// TIA Portal V21 export
FUNCTION_BLOCK "Inputs_FB"   // FB100, LAD
{ S7_Optimized_Access := 'TRUE' }
// stored: AutoNumber false, MemoryReserve 100, SetENOAutomatically false
   VAR
      ResetEdge { ExternalAccessible := 'False'; ExternalVisible := 'False'; ExternalWritable := 'False'} : Bool;
      TankLevel { ExternalAccessible := 'False'; ExternalVisible := 'False'; ExternalWritable := 'False'} : Array[1..2] of "AnalogInput";
   END_VAR
   VAR_TEMP   // added for the SCL form of the ladder/FBD networks
      _w1 : Bool;
      _w2 : Bool;
   END_VAR
BEGIN

REGION Network 1: === General
END_REGION

REGION Network 2: Emergency stop
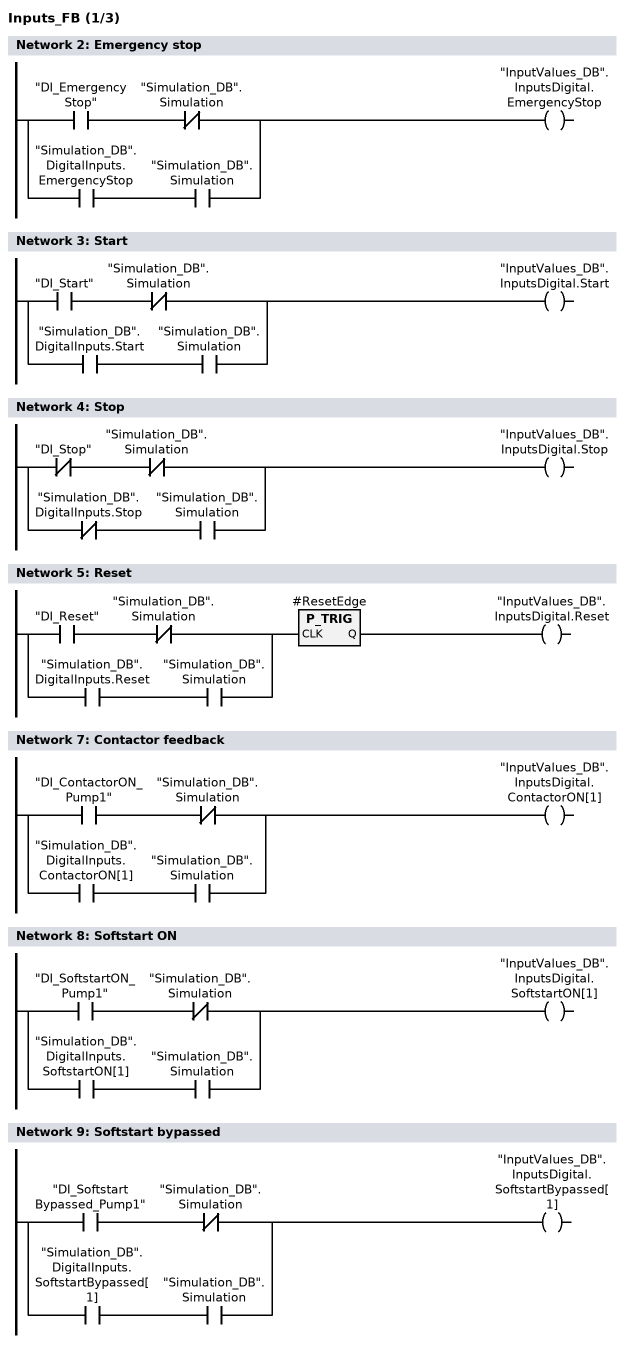
   RUNG wire#powerrail
      Contact( "DI_EmergencyStop" )
      I_Contact( "Simulation_DB".Simulation )
      wire#w1
      Coil( "InputValues_DB".InputsDigital.EmergencyStop )
   END_RUNG
   RUNG wire#powerrail
      Contact( "Simulation_DB".DigitalInputs.EmergencyStop )
      Contact( "Simulation_DB".Simulation )
   END_RUNG wire#w1
   // the same network as SCL:
   "InputValues_DB".InputsDigital.EmergencyStop := ("DI_EmergencyStop" AND NOT "Simulation_DB".Simulation) OR ("Simulation_DB".DigitalInputs.EmergencyStop AND "Simulation_DB".Simulation);
END_REGION

REGION Network 3: Start
   RUNG wire#powerrail
      Contact( "DI_Start" )
      I_Contact( "Simulation_DB".Simulation )
      wire#w1
      Coil( "InputValues_DB".InputsDigital.Start )
   END_RUNG
   RUNG wire#powerrail
      Contact( "Simulation_DB".DigitalInputs.Start )
      Contact( "Simulation_DB".Simulation )
   END_RUNG wire#w1
   // the same network as SCL:
   "InputValues_DB".InputsDigital.Start := ("DI_Start" AND NOT "Simulation_DB".Simulation) OR ("Simulation_DB".DigitalInputs.Start AND "Simulation_DB".Simulation);
END_REGION

REGION Network 4: Stop
   RUNG wire#powerrail
      I_Contact( "DI_Stop" )
      I_Contact( "Simulation_DB".Simulation )
      wire#w1
      Coil( "InputValues_DB".InputsDigital.Stop )
   END_RUNG
   RUNG wire#powerrail
      I_Contact( "Simulation_DB".DigitalInputs.Stop )
      Contact( "Simulation_DB".Simulation )
   END_RUNG wire#w1
   // the same network as SCL:
   "InputValues_DB".InputsDigital.Stop := (NOT "DI_Stop" AND NOT "Simulation_DB".Simulation) OR (NOT "Simulation_DB".DigitalInputs.Stop AND "Simulation_DB".Simulation);
END_REGION

REGION Network 5: Reset
   RUNG wire#powerrail
      Contact( "DI_Reset" )
      I_Contact( "Simulation_DB".Simulation )
      wire#w1
      P_Trig( #ResetEdge )
      Coil( "InputValues_DB".InputsDigital.Reset )
   END_RUNG
   RUNG wire#powerrail
      Contact( "Simulation_DB".DigitalInputs.Reset )
      Contact( "Simulation_DB".Simulation )
   END_RUNG wire#w1
   // the same network as SCL:
   #_w1 := ("DI_Reset" AND NOT "Simulation_DB".Simulation) OR ("Simulation_DB".DigitalInputs.Reset AND "Simulation_DB".Simulation);
   #_w2 := #_w1 AND NOT #ResetEdge;   // rising edge
   #ResetEdge := #_w1;
   "InputValues_DB".InputsDigital.Reset := #_w2;
END_REGION

REGION Network 6: === Pump 1
END_REGION

REGION Network 7: Contactor feedback
   RUNG wire#powerrail
      Contact( "DI_ContactorON_Pump1" )
      I_Contact( "Simulation_DB".Simulation )
      wire#w1
      Coil( "InputValues_DB".InputsDigital.ContactorON[1] )
   END_RUNG
   RUNG wire#powerrail
      Contact( "Simulation_DB".DigitalInputs.ContactorON[1] )
      Contact( "Simulation_DB".Simulation )
   END_RUNG wire#w1
   // the same network as SCL:
   "InputValues_DB".InputsDigital.ContactorON[1] := ("DI_ContactorON_Pump1" AND NOT "Simulation_DB".Simulation) OR ("Simulation_DB".DigitalInputs.ContactorON[1] AND "Simulation_DB".Simulation);
END_REGION

REGION Network 8: Softstart ON
   RUNG wire#powerrail
      Contact( "DI_SoftstartON_Pump1" )
      I_Contact( "Simulation_DB".Simulation )
      wire#w1
      Coil( "InputValues_DB".InputsDigital.SoftstartON[1] )
   END_RUNG
   RUNG wire#powerrail
      Contact( "Simulation_DB".DigitalInputs.SoftstartON[1] )
      Contact( "Simulation_DB".Simulation )
   END_RUNG wire#w1
   // the same network as SCL:
   "InputValues_DB".InputsDigital.SoftstartON[1] := ("DI_SoftstartON_Pump1" AND NOT "Simulation_DB".Simulation) OR ("Simulation_DB".DigitalInputs.SoftstartON[1] AND "Simulation_DB".Simulation);
END_REGION

REGION Network 9: Softstart bypassed
   RUNG wire#powerrail
      Contact( "DI_SoftstartBypassed_Pump1" )
      I_Contact( "Simulation_DB".Simulation )
      wire#w1
      Coil( "InputValues_DB".InputsDigital.SoftstartBypassed[1] )
   END_RUNG
   RUNG wire#powerrail
      Contact( "Simulation_DB".DigitalInputs.SoftstartBypassed[1] )
      Contact( "Simulation_DB".Simulation )
   END_RUNG wire#w1
   // the same network as SCL:
   "InputValues_DB".InputsDigital.SoftstartBypassed[1] := ("DI_SoftstartBypassed_Pump1" AND NOT "Simulation_DB".Simulation) OR ("Simulation_DB".DigitalInputs.SoftstartBypassed[1] AND "Simulation_DB".Simulation);
END_REGION

REGION Network 10: Softstart fault
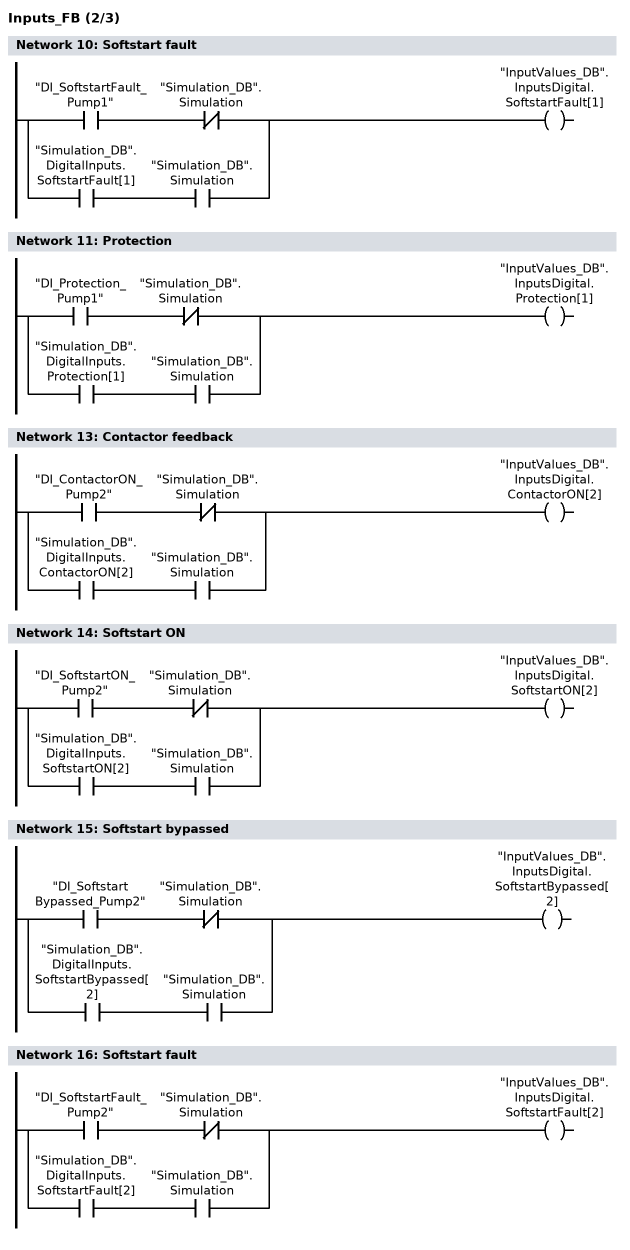
   RUNG wire#powerrail
      Contact( "DI_SoftstartFault_Pump1" )
      I_Contact( "Simulation_DB".Simulation )
      wire#w1
      Coil( "InputValues_DB".InputsDigital.SoftstartFault[1] )
   END_RUNG
   RUNG wire#powerrail
      Contact( "Simulation_DB".DigitalInputs.SoftstartFault[1] )
      Contact( "Simulation_DB".Simulation )
   END_RUNG wire#w1
   // the same network as SCL:
   "InputValues_DB".InputsDigital.SoftstartFault[1] := ("DI_SoftstartFault_Pump1" AND NOT "Simulation_DB".Simulation) OR ("Simulation_DB".DigitalInputs.SoftstartFault[1] AND "Simulation_DB".Simulation);
END_REGION

REGION Network 11: Protection
   RUNG wire#powerrail
      Contact( "DI_Protection_Pump1" )
      I_Contact( "Simulation_DB".Simulation )
      wire#w1
      Coil( "InputValues_DB".InputsDigital.Protection[1] )
   END_RUNG
   RUNG wire#powerrail
      Contact( "Simulation_DB".DigitalInputs.Protection[1] )
      Contact( "Simulation_DB".Simulation )
   END_RUNG wire#w1
   // the same network as SCL:
   "InputValues_DB".InputsDigital.Protection[1] := ("DI_Protection_Pump1" AND NOT "Simulation_DB".Simulation) OR ("Simulation_DB".DigitalInputs.Protection[1] AND "Simulation_DB".Simulation);
END_REGION

REGION Network 12: === Pump 2
END_REGION

REGION Network 13: Contactor feedback
   RUNG wire#powerrail
      Contact( "DI_ContactorON_Pump2" )
      I_Contact( "Simulation_DB".Simulation )
      wire#w1
      Coil( "InputValues_DB".InputsDigital.ContactorON[2] )
   END_RUNG
   RUNG wire#powerrail
      Contact( "Simulation_DB".DigitalInputs.ContactorON[2] )
      Contact( "Simulation_DB".Simulation )
   END_RUNG wire#w1
   // the same network as SCL:
   "InputValues_DB".InputsDigital.ContactorON[2] := ("DI_ContactorON_Pump2" AND NOT "Simulation_DB".Simulation) OR ("Simulation_DB".DigitalInputs.ContactorON[2] AND "Simulation_DB".Simulation);
END_REGION

REGION Network 14: Softstart ON
   RUNG wire#powerrail
      Contact( "DI_SoftstartON_Pump2" )
      I_Contact( "Simulation_DB".Simulation )
      wire#w1
      Coil( "InputValues_DB".InputsDigital.SoftstartON[2] )
   END_RUNG
   RUNG wire#powerrail
      Contact( "Simulation_DB".DigitalInputs.SoftstartON[2] )
      Contact( "Simulation_DB".Simulation )
   END_RUNG wire#w1
   // the same network as SCL:
   "InputValues_DB".InputsDigital.SoftstartON[2] := ("DI_SoftstartON_Pump2" AND NOT "Simulation_DB".Simulation) OR ("Simulation_DB".DigitalInputs.SoftstartON[2] AND "Simulation_DB".Simulation);
END_REGION

REGION Network 15: Softstart bypassed
   RUNG wire#powerrail
      Contact( "DI_SoftstartBypassed_Pump2" )
      I_Contact( "Simulation_DB".Simulation )
      wire#w1
      Coil( "InputValues_DB".InputsDigital.SoftstartBypassed[2] )
   END_RUNG
   RUNG wire#powerrail
      Contact( "Simulation_DB".DigitalInputs.SoftstartBypassed[2] )
      Contact( "Simulation_DB".Simulation )
   END_RUNG wire#w1
   // the same network as SCL:
   "InputValues_DB".InputsDigital.SoftstartBypassed[2] := ("DI_SoftstartBypassed_Pump2" AND NOT "Simulation_DB".Simulation) OR ("Simulation_DB".DigitalInputs.SoftstartBypassed[2] AND "Simulation_DB".Simulation);
END_REGION

REGION Network 16: Softstart fault
   RUNG wire#powerrail
      Contact( "DI_SoftstartFault_Pump2" )
      I_Contact( "Simulation_DB".Simulation )
      wire#w1
      Coil( "InputValues_DB".InputsDigital.SoftstartFault[2] )
   END_RUNG
   RUNG wire#powerrail
      Contact( "Simulation_DB".DigitalInputs.SoftstartFault[2] )
      Contact( "Simulation_DB".Simulation )
   END_RUNG wire#w1
   // the same network as SCL:
   "InputValues_DB".InputsDigital.SoftstartFault[2] := ("DI_SoftstartFault_Pump2" AND NOT "Simulation_DB".Simulation) OR ("Simulation_DB".DigitalInputs.SoftstartFault[2] AND "Simulation_DB".Simulation);
END_REGION

REGION Network 17: Protection
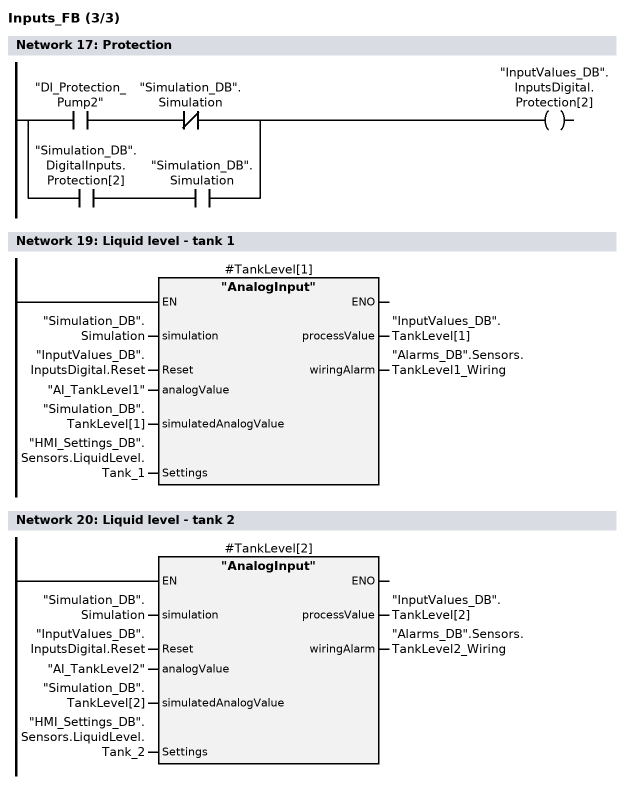
   RUNG wire#powerrail
      Contact( "DI_Protection_Pump2" )
      I_Contact( "Simulation_DB".Simulation )
      wire#w1
      Coil( "InputValues_DB".InputsDigital.Protection[2] )
   END_RUNG
   RUNG wire#powerrail
      Contact( "Simulation_DB".DigitalInputs.Protection[2] )
      Contact( "Simulation_DB".Simulation )
   END_RUNG wire#w1
   // the same network as SCL:
   "InputValues_DB".InputsDigital.Protection[2] := ("DI_Protection_Pump2" AND NOT "Simulation_DB".Simulation) OR ("Simulation_DB".DigitalInputs.Protection[2] AND "Simulation_DB".Simulation);
END_REGION

REGION Network 18: === Analog inputs
END_REGION

REGION Network 19: Liquid level - tank 1
   RUNG wire#powerrail
      #TankLevel[1](simulation := "Simulation_DB".Simulation, Reset := "InputValues_DB".InputsDigital.Reset, analogValue := "AI_TankLevel1", simulatedAnalogValue := "Simulation_DB".TankLevel[1], Settings := "HMI_Settings_DB".Sensors.LiquidLevel.Tank_1, processValue => "InputValues_DB".TankLevel[1], wiringAlarm => "Alarms_DB".Sensors.TankLevel1_Wiring)
   END_RUNG
   // the same network as SCL:
   #TankLevel[1](simulation := "Simulation_DB".Simulation,   // "AnalogInput"
                 Reset := "InputValues_DB".InputsDigital.Reset,
                 analogValue := "AI_TankLevel1",
                 simulatedAnalogValue := "Simulation_DB".TankLevel[1],
                 Settings := "HMI_Settings_DB".Sensors.LiquidLevel.Tank_1,
                 processValue => "InputValues_DB".TankLevel[1],
                 wiringAlarm => "Alarms_DB".Sensors.TankLevel1_Wiring);
END_REGION

REGION Network 20: Liquid level - tank 2
   RUNG wire#powerrail
      #TankLevel[2](simulation := "Simulation_DB".Simulation, Reset := "InputValues_DB".InputsDigital.Reset, analogValue := "AI_TankLevel2", simulatedAnalogValue := "Simulation_DB".TankLevel[2], Settings := "HMI_Settings_DB".Sensors.LiquidLevel.Tank_2, processValue => "InputValues_DB".TankLevel[2], wiringAlarm => "Alarms_DB".Sensors.TankLevel2_Wiring)
   END_RUNG
   // the same network as SCL:
   #TankLevel[2](simulation := "Simulation_DB".Simulation,   // "AnalogInput"
                 Reset := "InputValues_DB".InputsDigital.Reset,
                 analogValue := "AI_TankLevel2",
                 simulatedAnalogValue := "Simulation_DB".TankLevel[2],
                 Settings := "HMI_Settings_DB".Sensors.LiquidLevel.Tank_2,
                 processValue => "InputValues_DB".TankLevel[2],
                 wiringAlarm => "Alarms_DB".Sensors.TankLevel2_Wiring);
END_REGION
END_FUNCTION_BLOCK
